FUNCTION "LPMLV2022_ConfigureDisabledStatesCfg" : Void
TITLE = LPMLV2022_ConfigureDisabledStatesCfg
{ S7_Optimized_Access := 'TRUE' }
AUTHOR : APC_ERLF
FAMILY : OMAC
VERSION : 1.0
//Support: tech.team.motioncontrol@siemens.com
   VAR_INPUT
      Clearing : Bool;   // TRUE: Disable state Clearing
      Starting : Bool;   // TRUE: Disable state Starting
      Suspended : Bool;   // TRUE: Disable state Suspended
      Stopping : Bool;   // TRUE: Disable state Stopping
      Aborting : Bool;   // TRUE: Disable state Aborting
      Holding : Bool;   // TRUE: Disable state Holding
      Held : Bool;   // TRUE: Disable state Held
      Unholding : Bool;   // TRUE: Disable state Unholding
      Suspending : Bool;   // TRUE: Disable state Suspending
      Unsuspending : Bool;   // TRUE: Disable state Unsuspending
      Resetting : Bool;   // TRUE: Disable state Resetting
      Completing : Bool;   // TRUE: Disable state Completing
      Completed : Bool;   // TRUE: Disable state Completed
   END_VAR

   VAR_OUTPUT
      DisabledStatesCfg : DWord;   // Disabled states configuration for one unit mode. Bit locations within the DWORD value represent State numbers
   END_VAR


BEGIN
	REGION HEADER
	  //================================================================================
	  // SIEMENS AG
	  // (c)Copyright 2023 All Rights Reserved
	  //--------------------------------------------------------------------------------
	  // Library: LPMLV2022
	  // Tested with: S7-1211 with FW version V4.2, S7-1511-1 PN with FW version V2.6
	  // Engineering: TIA Portal V15.1
	  // Restrictions: -
	  // Requirements: S7-1200 FW 4.2 / S7-1500 FW 2.6
	  // Functionality: The function generates a DWord value which represents
	  //                the state configuration for one unit mode.
	  // Support: tech.team.motioncontrol@siemens.com
	  // Note: Parameter comments are only available in language 'English (United States)'
	  //--------------------------------------------------------------------------------
	  // Change log table:
	  // Version  Date        Expert in charge  Changes applied
	  // 01.00.00 28.02.2023  KT                First released version
	  //================================================================================
	END_REGION

	// Initialize states configuration
	#DisabledStatesCfg := 16#0000_0000;

	// Note: Stopped (.%X2), Idle (.%X4), Execute (.%X6) and Aborted (.%X9) are always present. They cannot be disabled

	// Set states configuration
	#DisabledStatesCfg.%X1  := #Clearing;
	#DisabledStatesCfg.%X3  := #Starting;
	#DisabledStatesCfg.%X5  := #Suspended;
	#DisabledStatesCfg.%X7  := #Stopping;
	#DisabledStatesCfg.%X8  := #Aborting;
	#DisabledStatesCfg.%X10 := #Holding;
	#DisabledStatesCfg.%X11 := #Held;
	#DisabledStatesCfg.%X12 := #Unholding;
	#DisabledStatesCfg.%X13 := #Suspending;
	#DisabledStatesCfg.%X14 := #Unsuspending;
	#DisabledStatesCfg.%X15 := #Resetting;
	#DisabledStatesCfg.%X16 := #Completing;
	#DisabledStatesCfg.%X17 := #Completed;
END_FUNCTION

